SUBAPPLICATION Uebung_010b9 (* Toggle Flip-Flop mit IE Button_A1 BT_STILL_HELD *)
  (* Standard: 61499-2; Description: Copyright (c) 2023 Meisterschulen am Ostbahnhof This program and the accompanying materials are made available under the terms of the Eclipse Public License 2.0 which is available at https://www.eclipse.org/legal/epl-2.0/ SPDX-License-Identifier: EPL-2.0 *)
  (* Version 1.0, 2023-10-23, Franz Höpfinger, Meisterschulen am Ostbahnhof *)
  IMPORT ButtonActivationCode::BT_STILL_HELD;
  IMPORT Uebungen::const::UT::DefaultPool::Button_A1;
  IMPORT logiBUS::io::DQ::logiBUS_DO::Output_Q1;
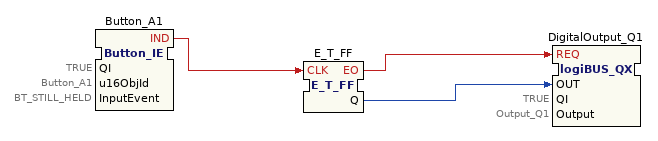
  (* BT_STILL_HELD wird alle 200ms wiederholt. ergibt also ein 400ms Blinker *)
  FBS
    DigitalOutput_Q1 : logiBUS::io::DQ::logiBUS_QX(QI := TRUE, Output := Output_Q1);
    Button_A1 : Button_IE(QI := TRUE, u16ObjId := Button_A1, InputEvent := BT_STILL_HELD);
    E_T_FF : iec61499::events::E_T_FF;
  END_FBS
  EVENT_CONNECTIONS
    Button_A1.IND TO E_T_FF.CLK;
    E_T_FF.EO TO DigitalOutput_Q1.REQ;
  END_CONNECTIONS
  DATA_CONNECTIONS
    E_T_FF.Q TO DigitalOutput_Q1.OUT;
  END_CONNECTIONS
END_SUBAPPLICATION
